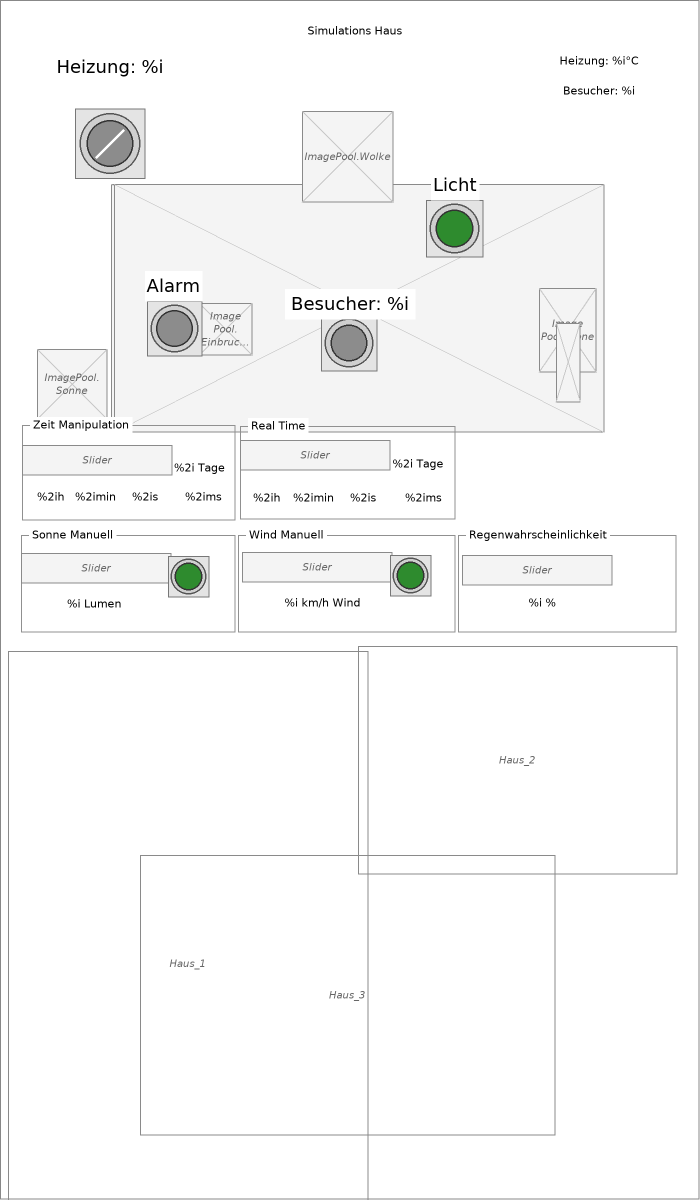
VISUALIZATION Simuliertes_Haus  // 700x1200
    Frame (8,651 360x625)
        shows Haus_1()
    Rectangle (24,44 652x371)
    Rectangle (24,44 652x371), colour variable: L_Himmel
        p2167032090: L_Himmel
    Image (111,184 490x248), image: ImagePool.Licht
        p84334746: HausSim.BildLicht
    Image (114,184 490x248), image: ImagePool.Haus
    Image (539,288 57x84), image: ImagePool.Krone
        p2858320360: L_Baum
    Image (556,323 24x79), image: ImagePool.Stamm
    Image (37,349 70x70), image: ImagePool.Sonne
        p2858320360: L_Sonnenstand
        p84334746: L_Sonne
    Image (199,303 53x52), image: ImagePool.Einbruch_grun
        p84334746: HausSim.L_EinbruchBild
    Image (302,111 91x91), image: ImagePool.Wolke
        p84334746: HausSim.WetterBild
    PushSwitch (147,300 55x57), variable: HausSim.Alarm_V, behaviour: TAP, style: Switch-PushSwitch-Gray
    Rectangle (145,271 57x30), "Alarm"
    Textfield (280,20 150x22), "Simulations Haus"
    Textfield (524,46 150x30), "Heizung: %i°C", text variable: HausSim.heizung_SIM
    Textfield (524,76 150x30), "Besucher: %i", text variable: HausSim.Besucher
    GroupBox (22,417 213x103), "Zeit Manipulation"
        Slider (0,28 150x30), variable: Zeit_Multiplikator, scale 0..4
        Textfield (41,65 65x30), "%2imin", text variable: _minute
        Textfield (90,65 66x30), "%2is", text variable: _sekunde
        Textfield (148,65 67x30), "%2ims", text variable: _mSekunde
        Textfield (-2,65 62x30), "%2ih", text variable: _stunde
        Textfield (149,36 61x30), "%2i Tage", text variable: day
    PushSwitch (426,200 57x57), variable: HausSim.L_Licht_V, behaviour: TAP, style: Switch-PushSwitch-Green
    Rectangle (431,170 48x30), "Licht", text variable: HausSim.Besucher
    GroupBox (240,418 215x101), "Real Time"
        Textfield (149,31 62x30), "%2i Tage", text variable: _Rday
        Slider (0,22 150x30), variable: Sin_manipulator, scale 0..3
        Textfield (41,65 65x30), "%2imin", text variable: _Rminute
        Textfield (90,65 66x30), "%2is", text variable: _Rsekunde
        Textfield (150,65 67x30), "%2ims", text variable: _RmSekunde
        Textfield (-4,65 62x30), "%2ih", text variable: _Rstunde
    GroupBox (458,527 218x105), "Regenwahrscheinlichkeit"
        Slider (4,28 150x30), variable: Regenwahrscheinlichkeit, scale 0..100
        Textfield (-18,61 205x30), "%i %", text variable: Regenwahrscheinlichkeit
    GroupBox (238,527 217x105), "Wind Manuell"
        Slider (4,25 150x30), variable: Wind_V, scale 0..200
        Textfield (-18,61 205x30), "%i km/h Wind", text variable: net_wind
        PushSwitch (152,28 41x41), variable: Wind_Auto_V, behaviour: TAP, style: Switch-PushSwitch-Green
    GroupBox (21,527 214x105), "Sonne Manuell"
        Slider (0,26 150x30), variable: Sonne_V, scale 100..2500
        Textfield (4,62 139x30), "%i Lumen", text variable: net_sonne
        PushSwitch (147,29 41x41), variable: Sonne_Auto_V, behaviour: TAP, style: Switch-PushSwitch-Green
    Frame (358,646 319x228)
        shows Haus_2()
    Frame (140,855 415x280)
        shows Haus_3()
    PushSwitch (321,314 56x58), variable: Sim_Haus_Glocke, behaviour: TAP, style: Switch-PushSwitch-Gray
    Rectangle (285,289 130x30), "Besucher: %i", text variable: HausSim.Besucher
    Potentiometer360 (75,105 70x77), variable: heizung_SIM, style: Potentiometer-Potentiometer360-Gray, scale format: %.1f, scale 14..30
    Rectangle (35,52 150x30), "Heizung: %i", text variable: heizung_SIM
END_VISUALIZATION

(* stored: Version 1.1.0.1, ProductVersion 3.1.4018.5
   Visu Simuliertes_Haus: Id {137e0316-b829-4758-93df-a9934f779ede} *)
